TYPE MBCommandsFrmCLC :
STRUCT
	//Commands from CLC  read at output register CLC master
	//state control enum type. 
	commands : StateMachineCommand;
	
	//P Q references. 
	ActivePowerReference : DINT;
	ReactivePowerReferecne: DINT;
	Heartbeat : DINT;
	ClrAlarm : DINT;
	ClrFault : DINT;
	
	
END_STRUCT
END_TYPE

(* stored: Version 1.1.0.1, ProductVersion 3.1.4024.11
   DUT MBCommandsFrmCLC: Id {ab42a186-6dc2-4c13-b087-70e5461a9097} *)
